PROGRAM MAIN
VAR
	Simulation		: FB_SIM;
	TypeControl		: FB_TypeControl;
	TypeUser		: U_Typeshift;
	Zone1			: FB_ZoneControl;
	Zone2			: FB_ZoneControl;
	Zone3			: FB_ZoneControl;	
	GenFault		: BOOL;
	userMain		: U_Main;	
	timing			: FB_Time;
	
	bInitDone		: BOOL;
	nCounter		: ULINT;
END_VAR

// Init
IF NOT bInitDone THEN
    // Init Settings
	Zone1.sZoneName := 'Zone A';
	Zone2.sZoneName := 'Zone B';
	Zone3.sZoneName := 'Zone X';
    bInitDone := TRUE;
END_IF


// Calls
timing();
Simulation();
userMain();
TypeControl();
Zone1(bError := Glob.bFault);
Zone2(bError := Glob.bFault);
Zone3(bError := Glob.bFault);


// Running Counter
nCounter	:=	nCounter + 1;

END_PROGRAM

(* stored: Version 1.1.0.1
   POU MAIN: Id {81cb7106-e41e-4ae5-8f62-d10f5f2cd019}, SpecialFunc None *)
